# EPICS substitutions: scllrfApp/Db/PRCextra.substitutions
file scllrfPRC.template
{
	{ NULL = NULL }
}

file scllrfCommon.template
{
	{ NULL = NULL }
}

file PRCwaves.template
{
pattern { N, EGU }
        { 0, V   }
        { 1, V   }
        { 2, V   }
        { 3, V   }
        { 4, V   }
        { 5, V   }
        { 6, V   }
        { 7, V   }
}

file PRCextra.template
{
	{ NULL = NULL }
}
